FUNCTION Convert_TIME_TO_USINT : BOOL
VAR_INPUT
	in : TIME;
	out : REFERENCE TO USINT;
END_VAR
VAR
	converted : USINT;
END_VAR

converted := TIME_TO_USINT(in);

IF (USINT_TO_TIME(converted) <> in) THEN
	RETURN;
END_IF

out := converted;
Convert_TIME_TO_USINT := TRUE;

END_FUNCTION

(* stored: Version 1.1.0.1, ProductVersion 3.1.4024.12
   POU Convert_TIME_TO_USINT: Id {c0360cbd-6fa4-4e8e-8c12-e02beed358ee}, SpecialFunc None *)
